Yaskawa INFORM job: SET0.JBI

/JOB
//NAME SET0
///FOLDERNAME FOLDER001
//POS
///NPOS 0,0,0,0,0,0
//INST
///DATE 2025/10/02 15:18
///ATTR SC,RW
///GROUP1 RB1
NOP
'SET TO 0
SET I066 0
SET I067 0
SET I068 0
SET I069 0
SET I070 0
SET I071 0
SET I072 0
SET I073 0
SET I074 0
SET I075 0
SET I076 0
SET I077 0
SET I078 0
SET I079 0
SET I080 0
SET I081 0
SET I082 0
SET I083 0
SET I065 0
SET I064 0
SET I063 0
SET I062 0
SET I061 0
SET I060 0
END
